FUNCTION_BLOCK Condition EXTENDS BaseConnector
VAR_INPUT
END_VAR
VAR_OUTPUT
END_VAR
VAR
	config		: ARRAY[0..99] OF ConditionConfig;
	result		: BOOL;
END_VAR

METHOD AndIs : REFERENCE TO Condition
VAR_INPUT
	symbol	: ANY;
END_VAR
END_METHOD

METHOD AndIsNot : Condition
VAR_INPUT
END_VAR
END_METHOD

METHOD Is : REFERENCE TO Condition
VAR_INPUT
	symbol	: ANY;
END_VAR
END_METHOD

METHOD IsNot : Condition
VAR_INPUT
END_VAR
END_METHOD

METHOD OrIs : Condition
VAR_INPUT
END_VAR
END_METHOD

METHOD OrIsNot : Condition
VAR_INPUT
END_VAR
END_METHOD

PROPERTY Satisfied : BOOL
GET
END_GET
END_PROPERTY

END_FUNCTION_BLOCK

(* stored: Version 1.1.0.1, ProductVersion 3.1.4024.11
   POU Condition: Id {1d377d48-3645-4a62-8c22-ed504447601c}, SpecialFunc None
   Method AndIs: Id {dafbc798-3481-496e-bdce-7334af149d57}
   Method AndIsNot: Id {8711eddd-8360-4b17-bf47-dc2bb0f47c6b}
   Method Is: Id {b29c744b-2cbb-408d-9901-5c0d667f11d2}
   Method IsNot: Id {eb1363f5-8800-437b-9dab-7e9f64ff6ef5}
   Method OrIs: Id {02886fb2-cdb6-4577-b186-b3f04d68735c}
   Method OrIsNot: Id {915f0eaf-e761-4267-b9b2-211fbfa70a1f}
   Property Satisfied: Id {3113431e-b25f-4d30-b220-6416ed2fcb70}
   Get Get: Id {4402da1e-296c-40c9-ad04-d77fde28b9ac} *)
